{attribute 'GeneratedUsingTerminal: EP9214-0023-0019'}
{attribute addProperty BoxType "EP9214-0023-0019"}
{attribute addProperty Id "DPO_Inputs_Channel_1AT %I*DPO_Inputs_Channel_BF408C5710DPO_Inputs_Channel_2AT %I*DPO_Inputs_Channel_BF408C5710DPO_Inputs_Channel_3AT %I*DPO_Inputs_Channel_BF408C5710DPO_Inputs_Channel_4AT %I*DPO_Inputs_Channel_BF408C5710DPO_Inputs_DeviceAT %I*DPO_Inputs_Device_9B08D91510DPO_Outputs_Channel_1AT %Q*DPO_Outputs_Channel_A459B36C4DPO_Outputs_Channel_2AT %Q*DPO_Outputs_Channel_A459B36C4DPO_Outputs_Channel_3AT %Q*DPO_Outputs_Channel_A459B36C4DPO_Outputs_Channel_4AT %Q*DPO_Outputs_Channel_A459B36C4DPO_Outputs_DeviceAT %Q*DPO_Outputs_Device_B673A3372WcStateAT %I*WcState_9091E0EB2InfoDataAT %I*InfoData_94A18F5E2"}
{attribute addProperty CRC "3303851285"}
{attribute addProperty Size "72"}
TYPE EP9214_C4ECC515 EXTENDS EtcSlaveTerminalBase_947E5A46 :
STRUCT
	{attribute addProperty Name "DPO_Inputs_Channel_1"}
	DPO_Inputs_Channel_1 : DPO_Inputs_Channel_BF408C57;
	{attribute addProperty Name "DPO_Inputs_Channel_2"}
	DPO_Inputs_Channel_2 : DPO_Inputs_Channel_BF408C57;
	{attribute addProperty Name "DPO_Inputs_Channel_3"}
	DPO_Inputs_Channel_3 : DPO_Inputs_Channel_BF408C57;
	{attribute addProperty Name "DPO_Inputs_Channel_4"}
	DPO_Inputs_Channel_4 : DPO_Inputs_Channel_BF408C57;
	{attribute addProperty Name "DPO_Inputs_Device"}
	DPO_Inputs_Device : DPO_Inputs_Device_9B08D915;
	{attribute addProperty Name "DPO_Outputs_Channel_1"}
	DPO_Outputs_Channel_1 : DPO_Outputs_Channel_A459B36C;
	{attribute addProperty Name "DPO_Outputs_Channel_2"}
	DPO_Outputs_Channel_2 : DPO_Outputs_Channel_A459B36C;
	{attribute addProperty Name "DPO_Outputs_Channel_3"}
	DPO_Outputs_Channel_3 : DPO_Outputs_Channel_A459B36C;
	{attribute addProperty Name "DPO_Outputs_Channel_4"}
	DPO_Outputs_Channel_4 : DPO_Outputs_Channel_A459B36C;
	{attribute addProperty Name "DPO_Outputs_Device"}
	DPO_Outputs_Device : DPO_Outputs_Device_B673A337;
	{attribute addProperty Name "WcState"}
	WcState : WcState_9091E0EB;
	{attribute addProperty Name "InfoData"}
	InfoData : InfoData_94A18F5E;
END_STRUCT
END_TYPE

(* stored: Version 1.2.0.0, ProductVersion 3.1.4024.9
   DUT EP9214_C4ECC515: Id {2de3f933-5c2d-4e80-82b4-ce6aa678dd52} *)
